INTERFACE I_AsyncCommandStateControl

METHOD PUBLIC Error
VAR_INPUT
	ErrorId : UDINT;
END_VAR
END_METHOD

METHOD PUBLIC Next
VAR_INPUT
END_VAR
END_METHOD

END_INTERFACE

(* stored: Version 1.1.0.1, ProductVersion 3.1.4024.12
   Itf I_AsyncCommandStateControl: Id {3b788fe5-63f3-0d48-2638-efc641ec0e6e}
   Method Error: Id {94ebc6b2-792e-08ca-2569-ff339b293157}
   Method Next: Id {82767363-400f-0977-1931-109037641119} *)
